FUNCTION_BLOCK FB_ObjCollectIterator
VAR_INPUT
	pInitNode : POINTER TO FB_ObjCollectionNode;
END_VAR
VAR_OUTPUT
	pNode : POINTER TO FB_ObjCollectionNode;
END_VAR
VAR
END_VAR

pNode := pInitNode;

METHOD M_Increment
VAR_INPUT
END_VAR
IF pNode > 0 AND_THEN pNode^.pNext > 0 THEN
	pNode := pNode^.pNext;
ELSE
	pNode := 0;
END_IF
END_METHOD

END_FUNCTION_BLOCK

(* stored: Version 1.1.0.1, ProductVersion 3.1.4022.12
   POU FB_ObjCollectIterator: Id {d9cb6f1a-c715-4c81-9454-8899f965b354}, SpecialFunc None
   Method M_Increment: Id {1d20ed23-7470-4aec-ab74-1a1cb0df0704} *)
